# EPICS StreamDevice protocol: smb100a-loc/smb100aApp/Db/smb100a.proto
# smb100a.proto for DMB100A Signal Generator
Terminator = LF;

get_id {
   out "*idn?";
   in "%#s";
}

get_ipaddr {
   out "syst:comm:netw:ipad?";
   in "%s";
}

get_freq {
   out "freq?";
   in "%f";
}

get_outp {
   out "outp?";
   in "%d";
}

get_out_pwr {
   out "pow?";
   in "%f";
}

set_freq {
   out "freq %f hz";
   @init { get_freq; }
 }

set_out_pwr {
   out "pow %f";
   @init { get_out_pwr; }
}

set_outp {
   out "outp %d";
   @init { get_outp; }
}

#
# LAN Interface Messages (do not change the instrument settings)
#
goto_local {
   out "&nren;&gtl";
}
goto_remote {
   out "&gtr";
}
not_remote_enbl {
   out "&nren";
}
dev_clear {
   out "&dcl";
}
local_lockout {
   out "&llo";
}
